FUNCTION F_CheckAlarm : BOOL
VAR_INPUT
	pTank : POINTER TO ST_Tank;
END_VAR
VAR
	fLevel : REAL := pTank^.fLevel;
	fTemperature : REAL := pTank^.fTemperature;
	fMaxTemperature : REAL := 80;
	fMaxLevelPercentage : REAL := 90;
END_VAR


IF pTank <> 0 THEN
	IF (fLevel > fMaxLevelPercentage) OR (fTemperature > fMaxTemperature )THEN
		F_CheckAlarm := TRUE;
	END_IF
END_IF

END_FUNCTION

(* stored: Version 1.1.0.1, ProductVersion 3.1.4024.16
   POU F_CheckAlarm: Id {4f67761f-9efd-4258-a475-4e091e8403c4}, SpecialFunc None *)
